{attribute addProperty BoxType "EL3423-0000-0016"}
{attribute addProperty Id "Reset_IntervalAT %Q*BOOL81"}
{attribute addProperty CRC "2882377394"}
{attribute addProperty SizeInBites "8"}
{attribute addProperty SizeInBytes "1"}
TYPE Interval_ABCD96B2 :
STRUCT
	{attribute addProperty Name "Reset_Interval"}
	Reset_Interval AT %Q* : BOOL;
END_STRUCT
END_TYPE

(* stored: Version 1.2.0.0, ProductVersion 3.1.4024.9
   DUT Interval_ABCD96B2: Id {d1898f7c-3917-4451-b1cb-026f29c9b92a} *)
